// TwinCAT 3 PLC project Untitled1
// ProgramVersion: 3.1.4024.0
// libraries:
//   Tc2_Standard, * (Beckhoff Automation GmbH)
//   Tc2_System, * (Beckhoff Automation GmbH)
//   Tc2_Utilities, * (Beckhoff Automation GmbH)
//   Tc3_Module, * (Beckhoff Automation GmbH)
// project tree:
//   DUTs/ E_EventType.TcDUT, ST_Event.TcDUT
//   / PlcTask.TcTTO
//   POUs/ EventLogger.TcPOU, FB_CsvPersistentEventStorage.TcPOU, I_PersistentEventStorage.TcIO, MAIN.TcPOU, UpdateEventTimestampWithSystemTime.TcPOU
// real-time tasks:
//   TASK PlcTask: cycle T#10ms, priority 20, ADS port 350

CONFIGURATION Untitled1
    RESOURCE PLC ON TwinCAT3
        TASK PlcTask(INTERVAL := T#10ms, PRIORITY := 20);
        PROGRAM MAIN WITH PlcTask : MAIN;
    END_RESOURCE
END_CONFIGURATION

// ---- DUTs/E_EventType.TcDUT
{attribute 'qualified_only'}
{attribute 'strict'}
{attribute 'to_string'}
TYPE E_EventType :
(
	Alarm := 0,
	Message := 1
);
END_TYPE

// ---- DUTs/ST_Event.TcDUT
TYPE ST_Event :
STRUCT
	eEventType : E_EventType;
	eEventSeverity : TcEventSeverity;
	nEventIdentity : UDINT;
	sEventText : STRING(255);
	dtTimeStamp : DATE_AND_TIME;
END_STRUCT
END_TYPE

// ---- POUs/I_PersistentEventStorage.TcIO
INTERFACE I_PersistentEventStorage

METHOD StoreEvent
VAR_INPUT
	stEvent : ST_Event;
END_VAR
//这个interface中只描述了存在这样一个方法，但是没有该方法具体如何操作的细节
END_METHOD

END_INTERFACE

// ---- POUs/MAIN.TcPOU
PROGRAM MAIN
VAR
	//stThisIsOurFirstInstanceOfStructure : ST_Event;
	bBoolean : BOOL := FALSE;
	
	eEventType1 : E_EventType := E_EventType.Alarm;
	eEventSeverity1 : TcEventSeverity := TcEventSeverity.Error;
	nEventIdentity1 : UDINT := 42;
	sEventText1 : STRING(255) := 'This is a scary event';
	

	CsvPersistentEventStorage : FB_CsvPersistentEventStorage;
	EventLogger : EventLogger(CsvPersistentEventStorage); //传递init所需要的参数
END_VAR

//IF NOT bBoolean THEN
	//UpdateEventTimestampWithSystemTime(stEvent := stThisIsOurFirstInstanceOfStructure);
	//bBoolean := TRUE;
//END_IF
IF bBoolean THEN
	EventLogger.AddEvent(eEventType := eEventType1,eEventSeverity1,nEventIdentity1,sEventText1);
	bBoolean := FALSE;
END_IF

CsvPersistentEventStorage();

END_PROGRAM

// ---- POUs/FB_CsvPersistentEventStorage.TcPOU
FUNCTION_BLOCK FB_CsvPersistentEventStorage IMPLEMENTS I_PersistentEventStorage
VAR
	eWriteState : (FILE_OPEN_TRIGGER, FILE_OPEN, WAIT_FOR_EVENT, WRITE_EVENT_TRIGGER, WRITE_EVENT, FILE_CLOSE_TRIGGER, FILE_CLOSE, ERROR);
	fb_FileOpen : FB_FileOpen := (sPathName := 'D:\Events.log', nMode := FOPEN_MODETEXT OR FOPEN_MODEAPPEND);
	fb_FilePuts : FB_FilePuts;
	fb_FileClose : FB_FileClose;
	stEventWrittenToFile : ST_event;
	Csvstring : T_MaxString;
END_VAR

CASE eWriteState OF
	
	FILE_OPEN_TRIGGER :
		fb_FileOpen(bExecute := TRUE) ;
		eWriteState := FILE_OPEN;
	FILE_OPEN :
		fb_FileOpen(bExecute := FALSE);
		IF fb_FileOpen.bError THEN
			eWriteState := ERROR;
		ELSIF NOT fb_FileOpen.bBusy AND fb_FileOpen.hFile <> 0 THEN
			eWriteState := WAIT_FOR_EVENT;
		END_IF
		
	WAIT_FOR_EVENT :
		// do not do anything
	WRITE_EVENT_TRIGGER:
		Csvstring := CreateCsvString(stEvent := stEventWrittenToFile);
		fb_FilePuts(bExecute := TRUE,
					sLine := Csvstring,
					hFile := fb_FileOpen.hFile);
		eWriteState := WRITE_EVENT;
	WRITE_EVENT : 
		fb_FilePuts(bExecute := FALSE);
		IF fb_FilePuts.bError THEN
			eWriteState := ERROR;
		ELSIF NOT fb_FilePuts.bBusy THEN
			eWriteState := WAIT_FOR_EVENT;
		END_IF
	
	FILE_CLOSE_TRIGGER :
		fb_FileClose(bExecute := TRUE,
					hFile := fb_FileOpen.hFile);
		eWriteState := FILE_CLOSE;
		
	FILE_CLOSE :
		fb_FileClose(bExecute := FALSE);
		IF fb_FileClose.bError THEN
			eWriteState := ERROR;
		ELSIF NOT fb_FileClose.bBusy THEN
			eWriteState := FILE_OPEN_TRIGGER;
		END_IF
	ERROR :
		// do nothing!
	
END_CASE

METHOD PRIVATE CreateCsvString : T_MaxString
VAR_INPUT
	stEvent : REFERENCE TO ST_Event;
END_VAR

VAR
	TempString : T_MaxString;
END_VAR
TempString := TO_STRING(stEvent.eEventType);
TempString := CONCAT(STR1 := TempString, STR2 := ',');
TempString := CONCAT(STR1 := TempString, STR2 := TO_STRING(stEvent.eEventSeverity));
TempString := CONCAT(STR1 := TempString, STR2 := ',');
TempString := CONCAT(STR1 := TempString, STR2 := TO_STRING(stEvent.nEventIdentity));
TempString := CONCAT(STR1 := TempString, STR2 := ',');
TempString := CONCAT(STR1 := TempString, STR2 := stEvent.sEventText);
TempString := CONCAT(STR1 := TempString, STR2 := ',');
TempString := CONCAT(STR1 := TempString, STR2 := TO_STRING(stEvent.dtTimeStamp));
TempString := CONCAT(STR1 := TempString, STR2 := '$n');

CreateCsvString := TempString;
END_METHOD

{warning '添加方法实现'}
METHOD StoreEvent
VAR_INPUT
	stEvent	: ST_Event;
END_VAR
//Here is where the csvwritting to be done
IF eWriteState = WAIT_FOR_EVENT THEN
	eWriteState := WRITE_EVENT_TRIGGER;
	stEventWrittenToFile := stEvent;
END_IF
END_METHOD

END_FUNCTION_BLOCK

// ---- POUs/EventLogger.TcPOU
FUNCTION_BLOCK PUBLIC EventLogger
VAR
	EventBuffer : ARRAY[1..MAXIMUM_SIZE_OF_EVENT_BUFFER] OF ST_Event; 
	CurrentEventBufferIndex : INT := 0;    
	
	_PersistentEventStorage : I_PersistentEventStorage; // 声明接口类型的变量
END_VAR
VAR CONSTANT
	MAXIMUM_SIZE_OF_EVENT_BUFFER : INT := 100;
END_VAR

METHOD PUBLIC AddEvent : BOOL
VAR_INPUT
	eEventType : E_EventType;
	eEventSeverity : TcEventSeverity;
	nEventIdentity : UDINT;
	sEventText : STRING(255);
END_VAR
IF NOT IsEventBufferFull() THEN
	CurrentEventBufferIndex := CurrentEventBufferIndex + 1;
	EventBuffer[CurrentEventBufferIndex].eEventType := eEventType;
	EventBuffer[CurrentEventBufferIndex].eEventSeverity := eEventSeverity;
	EventBuffer[CurrentEventBufferIndex].nEventIdentity := nEventIdentity;
	EventBuffer[CurrentEventBufferIndex].sEventText := sEventText;
	UpdateEventTimestampWithSystemTime(stEvent := EventBuffer[CurrentEventBufferIndex]);
	AddEvent := TRUE;
ELSE
	AddEvent := FALSE;
END_IF


//Here we want to store the event persistnetly by a reference
_PersistentEventStorage.StoreEvent(stEvent := EventBuffer[CurrentEventBufferIndex]);
END_METHOD

METHOD FB_init : BOOL
VAR_INPUT
	bInitRetains : BOOL; // if TRUE, the retain variables are initialized (warm start / cold start)
	bInCopyCode : BOOL;  // if TRUE, the instance afterwards gets moved into the copy code (online change)
	iPersistentEventStorage : I_PersistentEventStorage;
END_VAR
_PersistentEventStorage := iPersistentEventStorage; //给EventLogger中的内部变量赋值
END_METHOD

METHOD PRIVATE IsEventBufferFull : BOOL
IF (CurrentEventBufferIndex + 1) > MAXIMUM_SIZE_OF_EVENT_BUFFER THEN
	IsEventBufferFull := TRUE;
ELSE
	ISEventBufferFull := FALSE;
END_IF
END_METHOD

END_FUNCTION_BLOCK

// ---- POUs/UpdateEventTimestampWithSystemTime.TcPOU
FUNCTION UpdateEventTimestampWithSystemTime
VAR_INPUT
	stEvent : REFERENCE TO ST_Event;
	
END_VAR
VAR
	//fGetSystemTime : F_GetSystemTime; //实例化
	(*stFileTime : FILETIME64_TO_DT; //实例化，需要再reference中加入相关引用*)
	timeAsFileTime : T_FILETIME64;
	(*timeAsDT : DT;*)
END_VAR

timeAsFileTime := F_GetSystemTime();
stEvent.dtTimeStamp := FILETIME64_TO_DT(timeAsFileTime);

END_FUNCTION
